{attribute 'qualified_only'}
VAR_GLOBAL
	intDataToCSVINT		: INT;
	realDataToCSVREAL	: REAL;
END_VAR

(* stored: Version 1.1.0.1, ProductVersion 3.1.4024.11
   GVL csv_DB: Id {787faa80-4903-47a7-b09a-554280bd88f3} *)
